// TIA Portal V18 export
FUNCTION "select_remote" : Void   // FC36, FBD
{ S7_Optimized_Access := 'TRUE' }
VERSION : 0.1
// stored: AutoNumber true, IsIECCheckEnabled false, SetENOAutomatically false, UDAEnableTagReadback false
   VAR_INPUT
      MD_AUtO : Bool;
      MD_DESK : Bool;
      MD_RC : Bool;
      MD_RC_override : Bool;
      Joystick : Real;
      speed_RCfast : Real;
      speed_RCOverride : Real;
   END_VAR
   VAR_OUTPUT
      speed : Real;
   END_VAR
   VAR_IN_OUT
      m_AUTO : Bool;
      m_MAN : Bool;
      m_override : Bool;
   END_VAR
   VAR_TEMP
      slow_speed_static : Real;
      fast_speed_static : Real;
   END_VAR
BEGIN

REGION Network 2
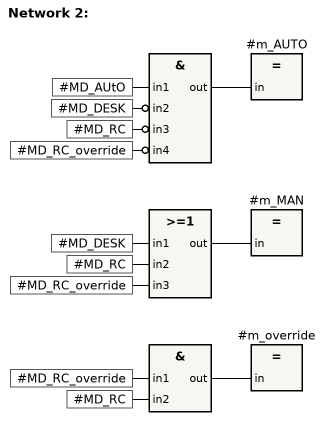
   #m_AUTO := #MD_AUtO AND NOT #MD_DESK AND NOT #MD_RC AND NOT #MD_RC_override;
   #m_MAN := #MD_DESK OR #MD_RC OR #MD_RC_override;
   #m_override := #MD_RC_override AND #MD_RC;
END_REGION
END_FUNCTION
